{attribute 'GeneratedUsingTerminal: EL6688-0000-0016'}
{attribute addProperty BoxType "EL6688-0000-0016"}
{attribute addProperty Id "EtcSlaveTerminalBaseSYNC_InputsAT %I*SYNC_Inputs_971453DD4WcStateAT %I*WcState_9091E0EB2InfoDataAT %I*InfoData_BEF6B88E18"}
{attribute addProperty CRC "2882602009"}
{attribute addProperty Size "24"}
TYPE EL6688_ABD10419 EXTENDS EtcSlaveTerminalBase :
STRUCT
	{attribute addProperty Name "SYNC_Inputs"}
	SYNC_Inputs : SYNC_Inputs_971453DD;
	{attribute addProperty Name "WcState"}
	WcState : WcState_9091E0EB;
	{attribute addProperty Name "InfoData"}
	InfoData : InfoData_BEF6B88E;
END_STRUCT
END_TYPE

(* stored: Version 1.2.0.0, ProductVersion 3.1.4024.9
   DUT EL6688_ABD10419: Id {4e59a1b0-17aa-4da0-94b1-fb7e24934f2c} *)
